FUNCTION_BLOCK FB_SequenceRNDWTR_Main EXTENDS FB_SequenceBase

VAR
	bUseMainPump_A: BOOL := TRUE;  // this boolean is used to keep track of which of the two redudant pumps we should use
END_VAR

VAR_IN_OUT
	devices: ST_RNDWTRComponents;
END_VAR

METHOD FB_init : BOOL
VAR_INPUT
	bInitRetains : BOOL; // if TRUE, the retain variables are initialized (warm start / cold start)
	bInCopyCode : BOOL;  // if TRUE, the instance afterwards gets moved into the copy code (online change)
	
	
END_VAR
(*
		Here we set the order of things to command, what the commands should be, and also how much time to allow during and between steps
		Every component listed below becomes 'Enabled' at each step
*)
sSequenceName:= 'R&D Rooms Lab WTR Main Sequence';
sSequenceDescription := 'Main sequence for R&D water treatment system';
END_METHOD

METHOD populateSteps : ST_SequenceStep
VAR_INPUT
	
END_VAR
(*
		Here we set the order of things to command, what the commands should be, and also how much time to allow during and between steps
		Every component listed below becomes 'Enabled' at each step
*)
Step1.Device := devices.fbUnit_RO_EDI;
Step1.Command := E_DeviceState.ON;
Step1.StepMinDuration := T#0S; 
Step1.DelayUntilNextStep := T#0S;
Step1.WaitForAction := FALSE;
aSequenceSteps[1] :=   Step1;

(*
Step2.Device := devices.fbUnit_RO_EDI;
Step2.Command := E_DeviceState.ON;
Step2.StepMinDuration := T#0S; 
Step2.DelayUntilNextStep := T#0S;
Step2.WaitForAction := FALSE;
aSequenceSteps[2] :=   Step2;
*)


nNumberSequenceSteps := 1;  // use this number to limit the number of operations
updateVarIDs();

(*

				Step8.Component := devices.
				Step8.Command := E_DeviceState.
				Step8.StepMinDuration := T#5S; 
				Step8.DelayUntilNextStep := T#5S;
				Step8.WaitForAction := TRUE;
				aSequenceSteps[8] :=   Step8;
				
				
				Step9.Component := devices.
				Step9.Command := E_DeviceState.
				Step9.StepMinDuration := T#5S; 
				Step9.DelayUntilNextStep := T#5S;
				Step9.WaitForAction := TRUE;
				aSequenceSteps[9] :=   Step9;
				
				
				Step10.Component := devices.
				Step10.Command := E_DeviceState.
				Step10.StepMinDuration := T#5S; 
				Step10.DelayUntilNextStep := T#5S;
				Step10.WaitForAction := TRUE;
				aSequenceSteps[10] :=   Step10;
				
				
				Step11.Component := devices.
				Step11.Command := E_DeviceState.
				Step11.StepMinDuration := T#5S; 
				Step11.DelayUntilNextStep := T#5S;
				Step11.WaitForAction := TRUE;
				aSequenceSteps[11] :=   Step11;
				
				
				Step12.Component := devices.
				Step12.Command := E_DeviceState.
				Step12.StepMinDuration := T#5S; 
				Step12.DelayUntilNextStep := T#5S;
				Step12.WaitForAction := TRUE;
				aSequenceSteps[12] :=   Step12;
				
				
				Step13.Component := devices.
				Step13.Command := E_DeviceState.
				Step13.StepMinDuration := T#5S; 
				Step13.DelayUntilNextStep := T#5S;
				Step13.WaitForAction := TRUE;
				aSequenceSteps[13] :=   Step13;
				
				
				Step14.Component := devices.
				Step14.Command := E_DeviceState.
				Step14.StepMinDuration := T#5S; 
				Step14.DelayUntilNextStep := T#5S;
				Step14.WaitForAction := TRUE;
				aSequenceSteps[14] :=   Step14;
				
				
				Step15.Component := devices.
				Step15.Command := E_DeviceState.
				Step15.StepMinDuration := T#5S; 
				Step15.DelayUntilNextStep := T#5S;
				Step15.WaitForAction := TRUE;
				aSequenceSteps[15] :=   Step15;
				
				
				Step16.Component := devices.
				Step16.Command := E_DeviceState.
				Step16.StepMinDuration := T#5S; 
				Step16.DelayUntilNextStep := T#5S;
				Step16.WaitForAction := TRUE;
				aSequenceSteps[16] :=   Step16;
				
				
				Step17.Component := devices.
				Step17.Command := E_DeviceState.
				Step17.StepMinDuration := T#5S; 
				Step17.DelayUntilNextStep := T#5S;
				Step17.WaitForAction := TRUE;
				aSequenceSteps[17] :=   Step17;
				
				
				Step18.Component := devices.
				Step18.Command := E_DeviceState.
				Step18.StepMinDuration := T#5S; 
				Step18.DelayUntilNextStep := T#5S;
				Step18.WaitForAction := TRUE;
				aSequenceSteps[18] :=   Step18;
				
				
				Step19.Component := devices.
				Step19.Command := E_DeviceState.
				Step19.StepMinDuration := T#5S; 
				Step19.DelayUntilNextStep := T#5S;
				Step19.WaitForAction := TRUE;
				aSequenceSteps[19] :=   Step19;
				
				
				Step20.Component := devices.
				Step20.Command := E_DeviceState.
				Step20.StepMinDuration := T#5S; 
				Step20.DelayUntilNextStep := T#5S;
				Step20.WaitForAction := TRUE;
				aSequenceSteps[20] :=   Step20;
*)
END_METHOD

END_FUNCTION_BLOCK

(* stored: Version 1.1.0.1, ProductVersion 3.1.4024.12
   POU FB_SequenceRNDWTR_Main: Id {027cb155-2402-4013-97ce-85c2432e6b66}, SpecialFunc None
   Method FB_init: Id {1a14cd02-3b14-4c92-8bd5-e871b807c634}
   Method populateSteps: Id {c89e4253-8efe-48eb-9296-6cb385a19e15} *)
